INTERFACE ITcoEthercatMasterDevice

PROPERTY AllDataValid : BOOL
GET
END_GET
END_PROPERTY

PROPERTY DeviceHasSomeIssue : BOOL
GET
END_GET
END_PROPERTY

PROPERTY SomeDataInvalid : BOOL
GET
END_GET
END_PROPERTY

PROPERTY SomeSyncUnitHasSomeIssue : BOOL
GET
END_GET
END_PROPERTY

PROPERTY State : TcoEthercatMasterDeviceState
GET
END_GET
END_PROPERTY

END_INTERFACE

(* stored: Version 1.1.0.1, ProductVersion 3.1.4024.9
   Itf ITcoEthercatMasterDevice: Id {da9fd16c-1d6e-03e6-3cbe-f6bc17dd6168}
   Property AllDataValid: Id {1859ac70-6c32-02cd-2ba0-460b02301642}
   Get Get: Id {3e35ef17-d2fe-01cb-2cf0-d66d2c72d094}
   Property DeviceHasSomeIssue: Id {40065bea-8268-0c34-00d5-cb2329162aca}
   Get Get: Id {ad4e8e61-3413-0e48-28bc-e5cd44fe4cc4}
   Property SomeDataInvalid: Id {f4e422c5-45f7-0bbc-37e3-dc0f899b801a}
   Get Get: Id {97daddac-6bfb-0211-05c0-f8e057e382da}
   Property SomeSyncUnitHasSomeIssue: Id {a8cb1f5f-0e38-0872-383d-988009353fc9}
   Get Get: Id {b9969bc2-273c-0941-2bc5-604ee8c5c77d}
   Property State: Id {99bff1c0-5401-07ba-06c1-9a3fa3cd9c18}
   Get Get: Id {10aaa00b-83e1-091d-2949-098cf7ebc563} *)
